// TIA Portal V17 export
// export: Created 2024-08-29T18:23:47.0171751Z, ExportSetting WithDefaults, DisplayName Totally Integrated Automation Portal, DisplayVersion V17 Update 7, DisplayName TIA Portal Openness, DisplayVersion V17 Update 7, DisplayName TIA Portal Version Control Interface, DisplayVersion V17, DisplayName SINAMICS Startdrive Advanced, DisplayVersion V17 SP2, DisplayName SINAMICS Startdrive G110M, G120, G120C, G120D, G120P, G115D, DisplayVersion V17 SP2, DisplayName SINAMICS Startdrive G130, G150, S120, S150, SINAMICS MV, S210, DisplayVersion V17 SP2, DisplayName STEP 7 Professional, DisplayVersion V17 Update 7, DisplayName STEP 7 Safety, DisplayVersion V17 Update 6, DisplayName WinCC Advanced / Unified PC, DisplayVersion V17 Update 7
FUNCTION "dintToBool" : Void   // FC10, LAD
{ S7_Optimized_Access := 'TRUE' }
VERSION : 0.1
// stored: AutoNumber true, IsIECCheckEnabled false, SetENOAutomatically false, UDAEnableTagReadback false
BEGIN

REGION Network 1: A INPUTS STATUS
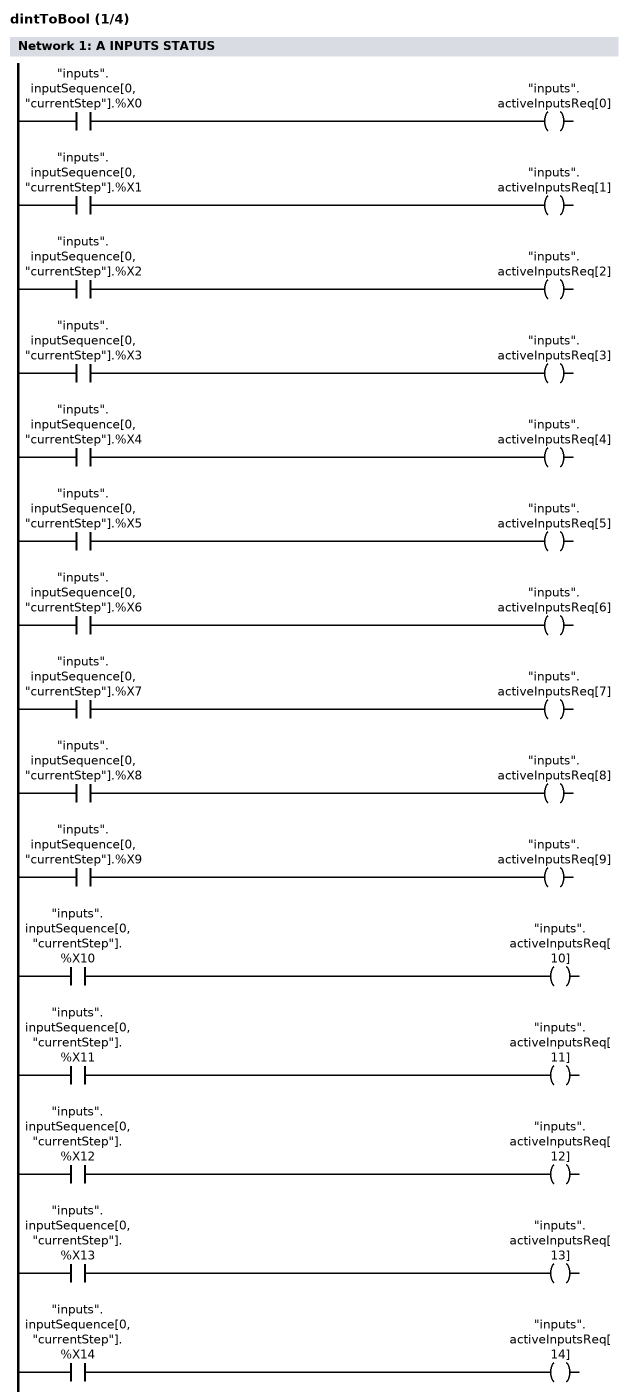
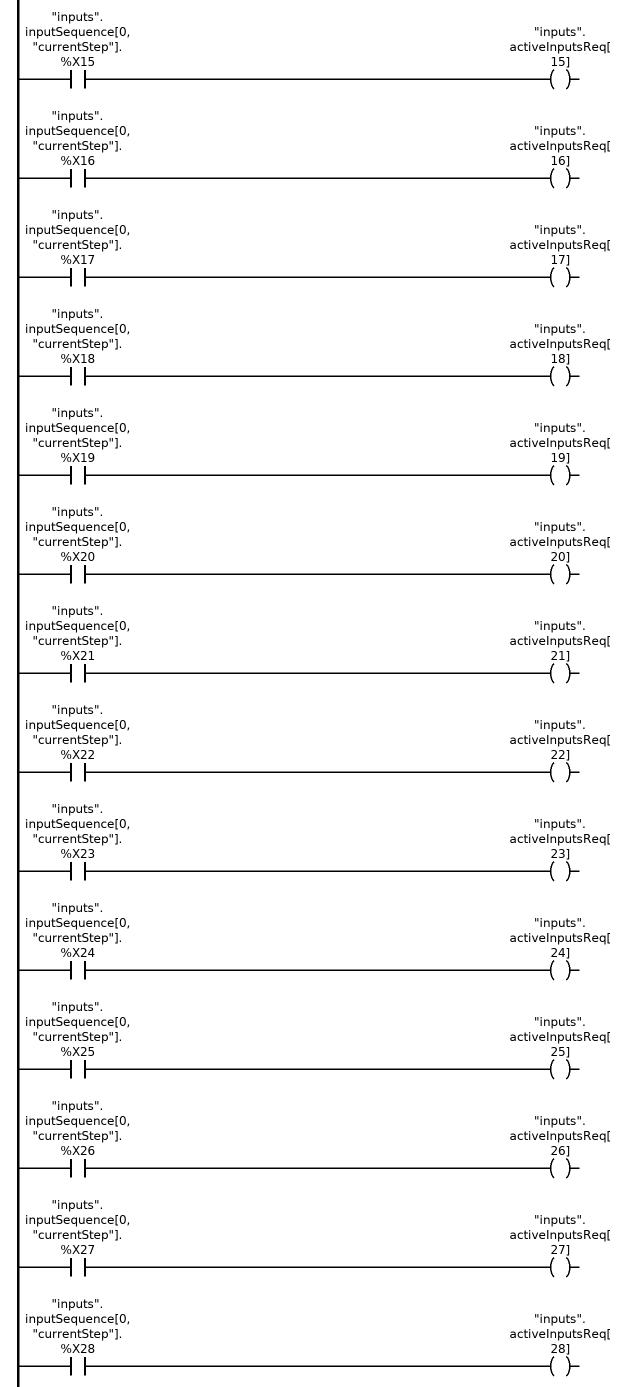
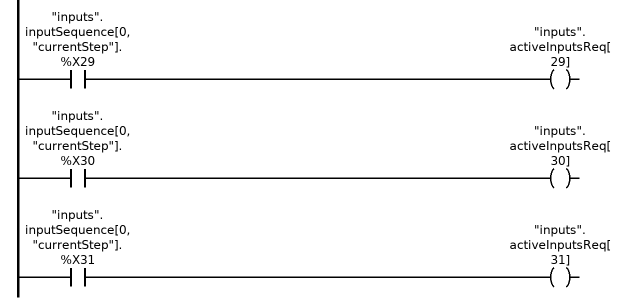
   RUNG wire#powerrail
      Contact( "inputs".inputSequence[0, "currentStep"].%X0 )
      Coil( "inputs".activeInputsReq[0] )
   END_RUNG
   RUNG wire#powerrail
      Contact( "inputs".inputSequence[0, "currentStep"].%X1 )
      Coil( "inputs".activeInputsReq[1] )
   END_RUNG
   RUNG wire#powerrail
      Contact( "inputs".inputSequence[0, "currentStep"].%X2 )
      Coil( "inputs".activeInputsReq[2] )
   END_RUNG
   RUNG wire#powerrail
      Contact( "inputs".inputSequence[0, "currentStep"].%X3 )
      Coil( "inputs".activeInputsReq[3] )
   END_RUNG
   RUNG wire#powerrail
      Contact( "inputs".inputSequence[0, "currentStep"].%X4 )
      Coil( "inputs".activeInputsReq[4] )
   END_RUNG
   RUNG wire#powerrail
      Contact( "inputs".inputSequence[0, "currentStep"].%X5 )
      Coil( "inputs".activeInputsReq[5] )
   END_RUNG
   RUNG wire#powerrail
      Contact( "inputs".inputSequence[0, "currentStep"].%X6 )
      Coil( "inputs".activeInputsReq[6] )
   END_RUNG
   RUNG wire#powerrail
      Contact( "inputs".inputSequence[0, "currentStep"].%X7 )
      Coil( "inputs".activeInputsReq[7] )
   END_RUNG
   RUNG wire#powerrail
      Contact( "inputs".inputSequence[0, "currentStep"].%X8 )
      Coil( "inputs".activeInputsReq[8] )
   END_RUNG
   RUNG wire#powerrail
      Contact( "inputs".inputSequence[0, "currentStep"].%X9 )
      Coil( "inputs".activeInputsReq[9] )
   END_RUNG
   RUNG wire#powerrail
      Contact( "inputs".inputSequence[0, "currentStep"].%X10 )
      Coil( "inputs".activeInputsReq[10] )
   END_RUNG
   RUNG wire#powerrail
      Contact( "inputs".inputSequence[0, "currentStep"].%X11 )
      Coil( "inputs".activeInputsReq[11] )
   END_RUNG
   RUNG wire#powerrail
      Contact( "inputs".inputSequence[0, "currentStep"].%X12 )
      Coil( "inputs".activeInputsReq[12] )
   END_RUNG
   RUNG wire#powerrail
      Contact( "inputs".inputSequence[0, "currentStep"].%X13 )
      Coil( "inputs".activeInputsReq[13] )
   END_RUNG
   RUNG wire#powerrail
      Contact( "inputs".inputSequence[0, "currentStep"].%X14 )
      Coil( "inputs".activeInputsReq[14] )
   END_RUNG
   RUNG wire#powerrail
      Contact( "inputs".inputSequence[0, "currentStep"].%X15 )
      Coil( "inputs".activeInputsReq[15] )
   END_RUNG
   RUNG wire#powerrail
      Contact( "inputs".inputSequence[0, "currentStep"].%X16 )
      Coil( "inputs".activeInputsReq[16] )
   END_RUNG
   RUNG wire#powerrail
      Contact( "inputs".inputSequence[0, "currentStep"].%X17 )
      Coil( "inputs".activeInputsReq[17] )
   END_RUNG
   RUNG wire#powerrail
      Contact( "inputs".inputSequence[0, "currentStep"].%X18 )
      Coil( "inputs".activeInputsReq[18] )
   END_RUNG
   RUNG wire#powerrail
      Contact( "inputs".inputSequence[0, "currentStep"].%X19 )
      Coil( "inputs".activeInputsReq[19] )
   END_RUNG
   RUNG wire#powerrail
      Contact( "inputs".inputSequence[0, "currentStep"].%X20 )
      Coil( "inputs".activeInputsReq[20] )
   END_RUNG
   RUNG wire#powerrail
      Contact( "inputs".inputSequence[0, "currentStep"].%X21 )
      Coil( "inputs".activeInputsReq[21] )
   END_RUNG
   RUNG wire#powerrail
      Contact( "inputs".inputSequence[0, "currentStep"].%X22 )
      Coil( "inputs".activeInputsReq[22] )
   END_RUNG
   RUNG wire#powerrail
      Contact( "inputs".inputSequence[0, "currentStep"].%X23 )
      Coil( "inputs".activeInputsReq[23] )
   END_RUNG
   RUNG wire#powerrail
      Contact( "inputs".inputSequence[0, "currentStep"].%X24 )
      Coil( "inputs".activeInputsReq[24] )
   END_RUNG
   RUNG wire#powerrail
      Contact( "inputs".inputSequence[0, "currentStep"].%X25 )
      Coil( "inputs".activeInputsReq[25] )
   END_RUNG
   RUNG wire#powerrail
      Contact( "inputs".inputSequence[0, "currentStep"].%X26 )
      Coil( "inputs".activeInputsReq[26] )
   END_RUNG
   RUNG wire#powerrail
      Contact( "inputs".inputSequence[0, "currentStep"].%X27 )
      Coil( "inputs".activeInputsReq[27] )
   END_RUNG
   RUNG wire#powerrail
      Contact( "inputs".inputSequence[0, "currentStep"].%X28 )
      Coil( "inputs".activeInputsReq[28] )
   END_RUNG
   RUNG wire#powerrail
      Contact( "inputs".inputSequence[0, "currentStep"].%X29 )
      Coil( "inputs".activeInputsReq[29] )
   END_RUNG
   RUNG wire#powerrail
      Contact( "inputs".inputSequence[0, "currentStep"].%X30 )
      Coil( "inputs".activeInputsReq[30] )
   END_RUNG
   RUNG wire#powerrail
      Contact( "inputs".inputSequence[0, "currentStep"].%X31 )
      Coil( "inputs".activeInputsReq[31] )
   END_RUNG
   // the same network as SCL:
   "inputs".activeInputsReq[0] := "inputs".inputSequence[0, "currentStep"].%X0;
   "inputs".activeInputsReq[1] := "inputs".inputSequence[0, "currentStep"].%X1;
   "inputs".activeInputsReq[2] := "inputs".inputSequence[0, "currentStep"].%X2;
   "inputs".activeInputsReq[3] := "inputs".inputSequence[0, "currentStep"].%X3;
   "inputs".activeInputsReq[4] := "inputs".inputSequence[0, "currentStep"].%X4;
   "inputs".activeInputsReq[5] := "inputs".inputSequence[0, "currentStep"].%X5;
   "inputs".activeInputsReq[6] := "inputs".inputSequence[0, "currentStep"].%X6;
   "inputs".activeInputsReq[7] := "inputs".inputSequence[0, "currentStep"].%X7;
   "inputs".activeInputsReq[8] := "inputs".inputSequence[0, "currentStep"].%X8;
   "inputs".activeInputsReq[9] := "inputs".inputSequence[0, "currentStep"].%X9;
   "inputs".activeInputsReq[10] := "inputs".inputSequence[0, "currentStep"].%X10;
   "inputs".activeInputsReq[11] := "inputs".inputSequence[0, "currentStep"].%X11;
   "inputs".activeInputsReq[12] := "inputs".inputSequence[0, "currentStep"].%X12;
   "inputs".activeInputsReq[13] := "inputs".inputSequence[0, "currentStep"].%X13;
   "inputs".activeInputsReq[14] := "inputs".inputSequence[0, "currentStep"].%X14;
   "inputs".activeInputsReq[15] := "inputs".inputSequence[0, "currentStep"].%X15;
   "inputs".activeInputsReq[16] := "inputs".inputSequence[0, "currentStep"].%X16;
   "inputs".activeInputsReq[17] := "inputs".inputSequence[0, "currentStep"].%X17;
   "inputs".activeInputsReq[18] := "inputs".inputSequence[0, "currentStep"].%X18;
   "inputs".activeInputsReq[19] := "inputs".inputSequence[0, "currentStep"].%X19;
   "inputs".activeInputsReq[20] := "inputs".inputSequence[0, "currentStep"].%X20;
   "inputs".activeInputsReq[21] := "inputs".inputSequence[0, "currentStep"].%X21;
   "inputs".activeInputsReq[22] := "inputs".inputSequence[0, "currentStep"].%X22;
   "inputs".activeInputsReq[23] := "inputs".inputSequence[0, "currentStep"].%X23;
   "inputs".activeInputsReq[24] := "inputs".inputSequence[0, "currentStep"].%X24;
   "inputs".activeInputsReq[25] := "inputs".inputSequence[0, "currentStep"].%X25;
   "inputs".activeInputsReq[26] := "inputs".inputSequence[0, "currentStep"].%X26;
   "inputs".activeInputsReq[27] := "inputs".inputSequence[0, "currentStep"].%X27;
   "inputs".activeInputsReq[28] := "inputs".inputSequence[0, "currentStep"].%X28;
   "inputs".activeInputsReq[29] := "inputs".inputSequence[0, "currentStep"].%X29;
   "inputs".activeInputsReq[30] := "inputs".inputSequence[0, "currentStep"].%X30;
   "inputs".activeInputsReq[31] := "inputs".inputSequence[0, "currentStep"].%X31;
END_REGION

REGION Network 2: MASK INPUTS STATUS
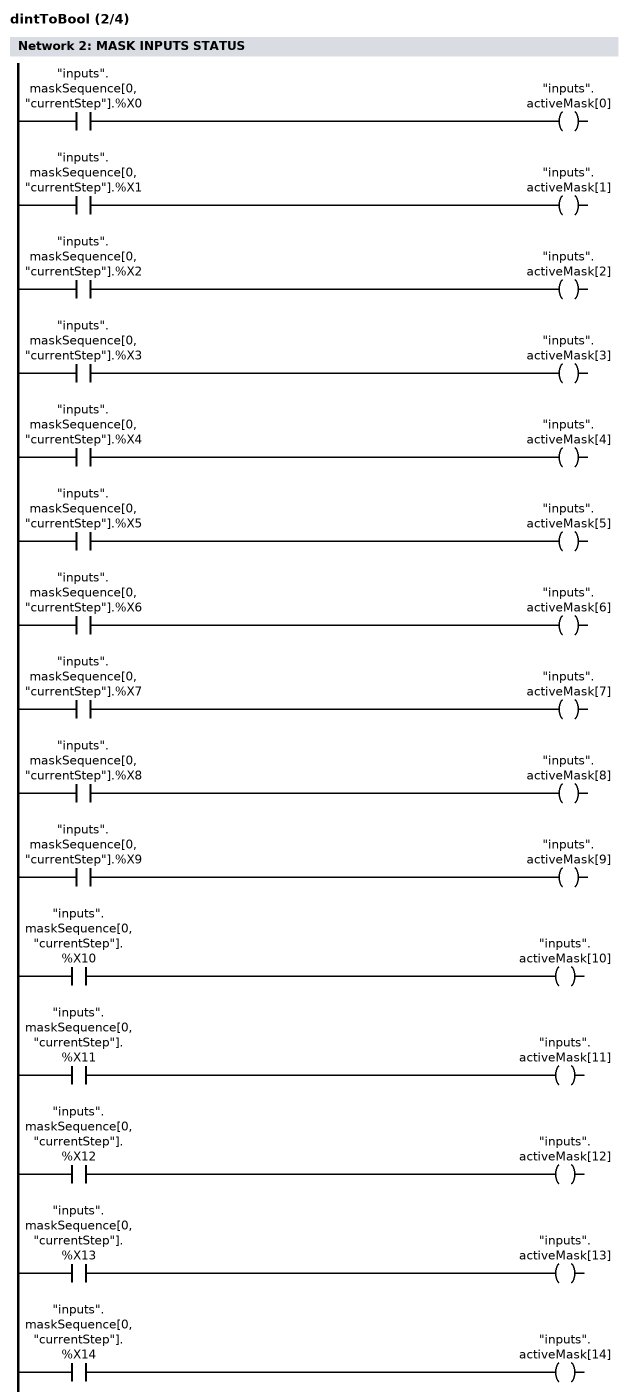
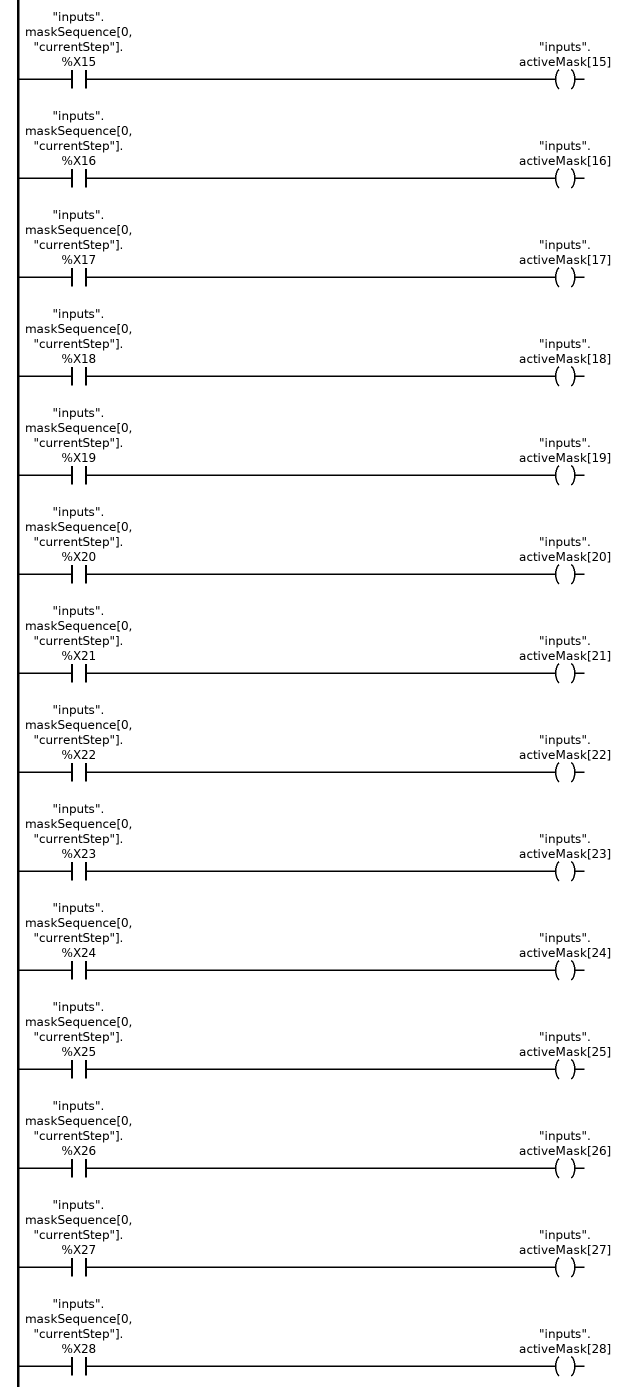
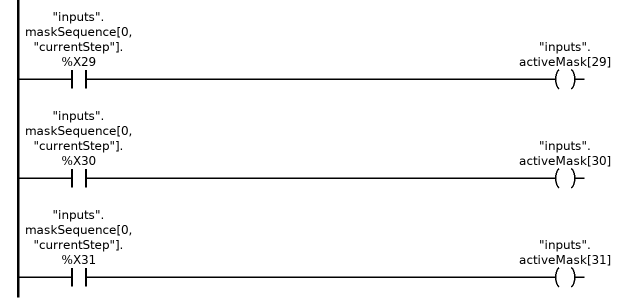
   RUNG wire#powerrail
      Contact( "inputs".maskSequence[0, "currentStep"].%X0 )
      Coil( "inputs".activeMask[0] )
   END_RUNG
   RUNG wire#powerrail
      Contact( "inputs".maskSequence[0, "currentStep"].%X1 )
      Coil( "inputs".activeMask[1] )
   END_RUNG
   RUNG wire#powerrail
      Contact( "inputs".maskSequence[0, "currentStep"].%X2 )
      Coil( "inputs".activeMask[2] )
   END_RUNG
   RUNG wire#powerrail
      Contact( "inputs".maskSequence[0, "currentStep"].%X3 )
      Coil( "inputs".activeMask[3] )
   END_RUNG
   RUNG wire#powerrail
      Contact( "inputs".maskSequence[0, "currentStep"].%X4 )
      Coil( "inputs".activeMask[4] )
   END_RUNG
   RUNG wire#powerrail
      Contact( "inputs".maskSequence[0, "currentStep"].%X5 )
      Coil( "inputs".activeMask[5] )
   END_RUNG
   RUNG wire#powerrail
      Contact( "inputs".maskSequence[0, "currentStep"].%X6 )
      Coil( "inputs".activeMask[6] )
   END_RUNG
   RUNG wire#powerrail
      Contact( "inputs".maskSequence[0, "currentStep"].%X7 )
      Coil( "inputs".activeMask[7] )
   END_RUNG
   RUNG wire#powerrail
      Contact( "inputs".maskSequence[0, "currentStep"].%X8 )
      Coil( "inputs".activeMask[8] )
   END_RUNG
   RUNG wire#powerrail
      Contact( "inputs".maskSequence[0, "currentStep"].%X9 )
      Coil( "inputs".activeMask[9] )
   END_RUNG
   RUNG wire#powerrail
      Contact( "inputs".maskSequence[0, "currentStep"].%X10 )
      Coil( "inputs".activeMask[10] )
   END_RUNG
   RUNG wire#powerrail
      Contact( "inputs".maskSequence[0, "currentStep"].%X11 )
      Coil( "inputs".activeMask[11] )
   END_RUNG
   RUNG wire#powerrail
      Contact( "inputs".maskSequence[0, "currentStep"].%X12 )
      Coil( "inputs".activeMask[12] )
   END_RUNG
   RUNG wire#powerrail
      Contact( "inputs".maskSequence[0, "currentStep"].%X13 )
      Coil( "inputs".activeMask[13] )
   END_RUNG
   RUNG wire#powerrail
      Contact( "inputs".maskSequence[0, "currentStep"].%X14 )
      Coil( "inputs".activeMask[14] )
   END_RUNG
   RUNG wire#powerrail
      Contact( "inputs".maskSequence[0, "currentStep"].%X15 )
      Coil( "inputs".activeMask[15] )
   END_RUNG
   RUNG wire#powerrail
      Contact( "inputs".maskSequence[0, "currentStep"].%X16 )
      Coil( "inputs".activeMask[16] )
   END_RUNG
   RUNG wire#powerrail
      Contact( "inputs".maskSequence[0, "currentStep"].%X17 )
      Coil( "inputs".activeMask[17] )
   END_RUNG
   RUNG wire#powerrail
      Contact( "inputs".maskSequence[0, "currentStep"].%X18 )
      Coil( "inputs".activeMask[18] )
   END_RUNG
   RUNG wire#powerrail
      Contact( "inputs".maskSequence[0, "currentStep"].%X19 )
      Coil( "inputs".activeMask[19] )
   END_RUNG
   RUNG wire#powerrail
      Contact( "inputs".maskSequence[0, "currentStep"].%X20 )
      Coil( "inputs".activeMask[20] )
   END_RUNG
   RUNG wire#powerrail
      Contact( "inputs".maskSequence[0, "currentStep"].%X21 )
      Coil( "inputs".activeMask[21] )
   END_RUNG
   RUNG wire#powerrail
      Contact( "inputs".maskSequence[0, "currentStep"].%X22 )
      Coil( "inputs".activeMask[22] )
   END_RUNG
   RUNG wire#powerrail
      Contact( "inputs".maskSequence[0, "currentStep"].%X23 )
      Coil( "inputs".activeMask[23] )
   END_RUNG
   RUNG wire#powerrail
      Contact( "inputs".maskSequence[0, "currentStep"].%X24 )
      Coil( "inputs".activeMask[24] )
   END_RUNG
   RUNG wire#powerrail
      Contact( "inputs".maskSequence[0, "currentStep"].%X25 )
      Coil( "inputs".activeMask[25] )
   END_RUNG
   RUNG wire#powerrail
      Contact( "inputs".maskSequence[0, "currentStep"].%X26 )
      Coil( "inputs".activeMask[26] )
   END_RUNG
   RUNG wire#powerrail
      Contact( "inputs".maskSequence[0, "currentStep"].%X27 )
      Coil( "inputs".activeMask[27] )
   END_RUNG
   RUNG wire#powerrail
      Contact( "inputs".maskSequence[0, "currentStep"].%X28 )
      Coil( "inputs".activeMask[28] )
   END_RUNG
   RUNG wire#powerrail
      Contact( "inputs".maskSequence[0, "currentStep"].%X29 )
      Coil( "inputs".activeMask[29] )
   END_RUNG
   RUNG wire#powerrail
      Contact( "inputs".maskSequence[0, "currentStep"].%X30 )
      Coil( "inputs".activeMask[30] )
   END_RUNG
   RUNG wire#powerrail
      Contact( "inputs".maskSequence[0, "currentStep"].%X31 )
      Coil( "inputs".activeMask[31] )
   END_RUNG
   // the same network as SCL:
   "inputs".activeMask[0] := "inputs".maskSequence[0, "currentStep"].%X0;
   "inputs".activeMask[1] := "inputs".maskSequence[0, "currentStep"].%X1;
   "inputs".activeMask[2] := "inputs".maskSequence[0, "currentStep"].%X2;
   "inputs".activeMask[3] := "inputs".maskSequence[0, "currentStep"].%X3;
   "inputs".activeMask[4] := "inputs".maskSequence[0, "currentStep"].%X4;
   "inputs".activeMask[5] := "inputs".maskSequence[0, "currentStep"].%X5;
   "inputs".activeMask[6] := "inputs".maskSequence[0, "currentStep"].%X6;
   "inputs".activeMask[7] := "inputs".maskSequence[0, "currentStep"].%X7;
   "inputs".activeMask[8] := "inputs".maskSequence[0, "currentStep"].%X8;
   "inputs".activeMask[9] := "inputs".maskSequence[0, "currentStep"].%X9;
   "inputs".activeMask[10] := "inputs".maskSequence[0, "currentStep"].%X10;
   "inputs".activeMask[11] := "inputs".maskSequence[0, "currentStep"].%X11;
   "inputs".activeMask[12] := "inputs".maskSequence[0, "currentStep"].%X12;
   "inputs".activeMask[13] := "inputs".maskSequence[0, "currentStep"].%X13;
   "inputs".activeMask[14] := "inputs".maskSequence[0, "currentStep"].%X14;
   "inputs".activeMask[15] := "inputs".maskSequence[0, "currentStep"].%X15;
   "inputs".activeMask[16] := "inputs".maskSequence[0, "currentStep"].%X16;
   "inputs".activeMask[17] := "inputs".maskSequence[0, "currentStep"].%X17;
   "inputs".activeMask[18] := "inputs".maskSequence[0, "currentStep"].%X18;
   "inputs".activeMask[19] := "inputs".maskSequence[0, "currentStep"].%X19;
   "inputs".activeMask[20] := "inputs".maskSequence[0, "currentStep"].%X20;
   "inputs".activeMask[21] := "inputs".maskSequence[0, "currentStep"].%X21;
   "inputs".activeMask[22] := "inputs".maskSequence[0, "currentStep"].%X22;
   "inputs".activeMask[23] := "inputs".maskSequence[0, "currentStep"].%X23;
   "inputs".activeMask[24] := "inputs".maskSequence[0, "currentStep"].%X24;
   "inputs".activeMask[25] := "inputs".maskSequence[0, "currentStep"].%X25;
   "inputs".activeMask[26] := "inputs".maskSequence[0, "currentStep"].%X26;
   "inputs".activeMask[27] := "inputs".maskSequence[0, "currentStep"].%X27;
   "inputs".activeMask[28] := "inputs".maskSequence[0, "currentStep"].%X28;
   "inputs".activeMask[29] := "inputs".maskSequence[0, "currentStep"].%X29;
   "inputs".activeMask[30] := "inputs".maskSequence[0, "currentStep"].%X30;
   "inputs".activeMask[31] := "inputs".maskSequence[0, "currentStep"].%X31;
END_REGION

REGION Network 3: B OUTPUTS STATUS
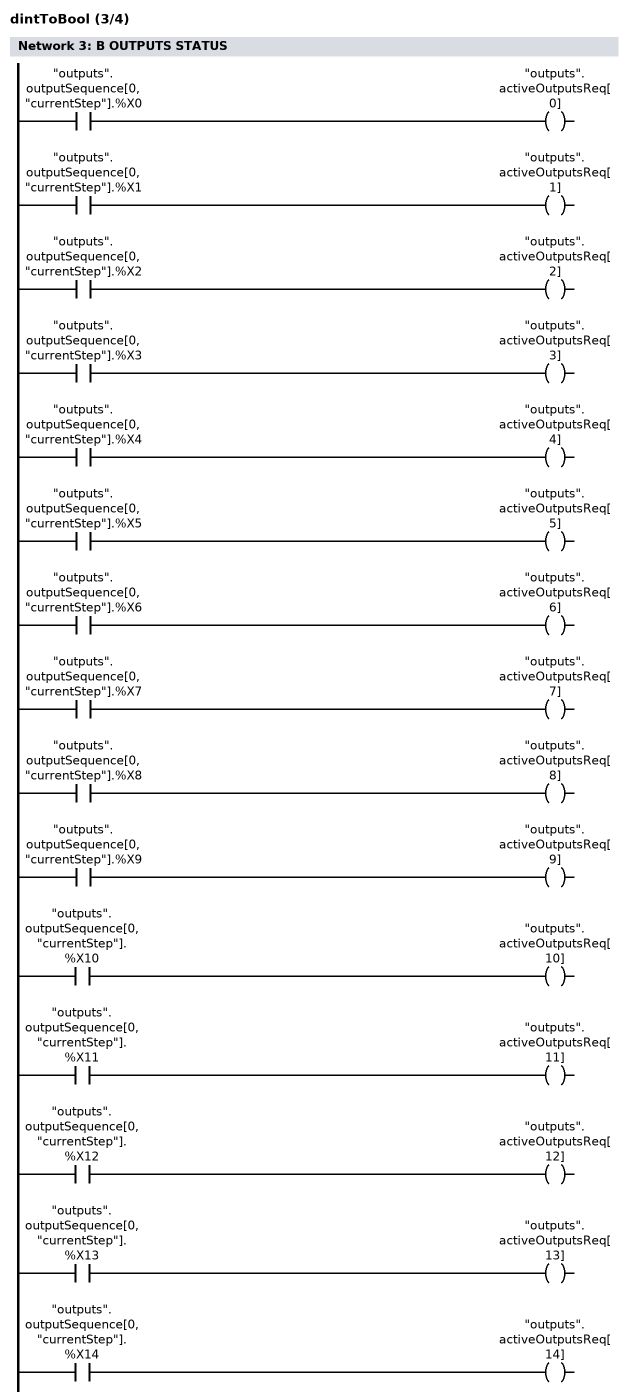
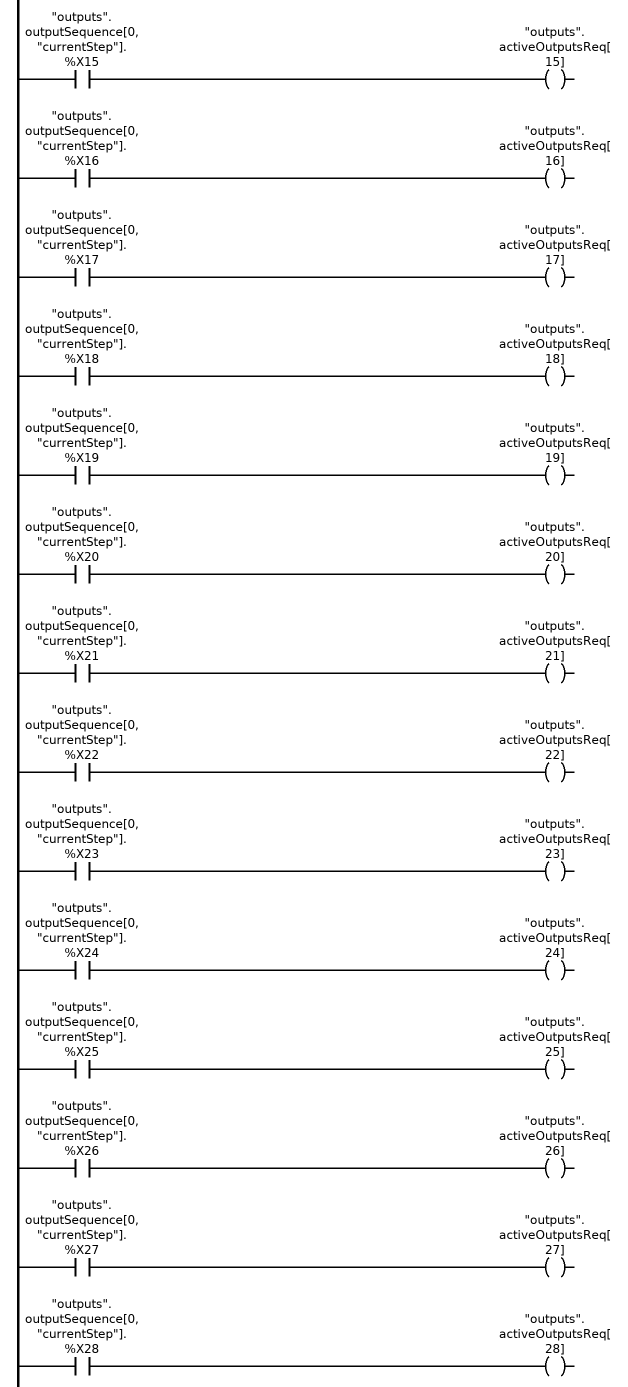
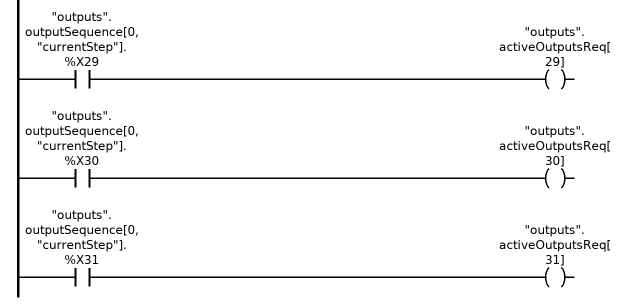
   RUNG wire#powerrail
      Contact( "outputs".outputSequence[0, "currentStep"].%X0 )
      Coil( "outputs".activeOutputsReq[0] )
   END_RUNG
   RUNG wire#powerrail
      Contact( "outputs".outputSequence[0, "currentStep"].%X1 )
      Coil( "outputs".activeOutputsReq[1] )
   END_RUNG
   RUNG wire#powerrail
      Contact( "outputs".outputSequence[0, "currentStep"].%X2 )
      Coil( "outputs".activeOutputsReq[2] )
   END_RUNG
   RUNG wire#powerrail
      Contact( "outputs".outputSequence[0, "currentStep"].%X3 )
      Coil( "outputs".activeOutputsReq[3] )
   END_RUNG
   RUNG wire#powerrail
      Contact( "outputs".outputSequence[0, "currentStep"].%X4 )
      Coil( "outputs".activeOutputsReq[4] )
   END_RUNG
   RUNG wire#powerrail
      Contact( "outputs".outputSequence[0, "currentStep"].%X5 )
      Coil( "outputs".activeOutputsReq[5] )
   END_RUNG
   RUNG wire#powerrail
      Contact( "outputs".outputSequence[0, "currentStep"].%X6 )
      Coil( "outputs".activeOutputsReq[6] )
   END_RUNG
   RUNG wire#powerrail
      Contact( "outputs".outputSequence[0, "currentStep"].%X7 )
      Coil( "outputs".activeOutputsReq[7] )
   END_RUNG
   RUNG wire#powerrail
      Contact( "outputs".outputSequence[0, "currentStep"].%X8 )
      Coil( "outputs".activeOutputsReq[8] )
   END_RUNG
   RUNG wire#powerrail
      Contact( "outputs".outputSequence[0, "currentStep"].%X9 )
      Coil( "outputs".activeOutputsReq[9] )
   END_RUNG
   RUNG wire#powerrail
      Contact( "outputs".outputSequence[0, "currentStep"].%X10 )
      Coil( "outputs".activeOutputsReq[10] )
   END_RUNG
   RUNG wire#powerrail
      Contact( "outputs".outputSequence[0, "currentStep"].%X11 )
      Coil( "outputs".activeOutputsReq[11] )
   END_RUNG
   RUNG wire#powerrail
      Contact( "outputs".outputSequence[0, "currentStep"].%X12 )
      Coil( "outputs".activeOutputsReq[12] )
   END_RUNG
   RUNG wire#powerrail
      Contact( "outputs".outputSequence[0, "currentStep"].%X13 )
      Coil( "outputs".activeOutputsReq[13] )
   END_RUNG
   RUNG wire#powerrail
      Contact( "outputs".outputSequence[0, "currentStep"].%X14 )
      Coil( "outputs".activeOutputsReq[14] )
   END_RUNG
   RUNG wire#powerrail
      Contact( "outputs".outputSequence[0, "currentStep"].%X15 )
      Coil( "outputs".activeOutputsReq[15] )
   END_RUNG
   RUNG wire#powerrail
      Contact( "outputs".outputSequence[0, "currentStep"].%X16 )
      Coil( "outputs".activeOutputsReq[16] )
   END_RUNG
   RUNG wire#powerrail
      Contact( "outputs".outputSequence[0, "currentStep"].%X17 )
      Coil( "outputs".activeOutputsReq[17] )
   END_RUNG
   RUNG wire#powerrail
      Contact( "outputs".outputSequence[0, "currentStep"].%X18 )
      Coil( "outputs".activeOutputsReq[18] )
   END_RUNG
   RUNG wire#powerrail
      Contact( "outputs".outputSequence[0, "currentStep"].%X19 )
      Coil( "outputs".activeOutputsReq[19] )
   END_RUNG
   RUNG wire#powerrail
      Contact( "outputs".outputSequence[0, "currentStep"].%X20 )
      Coil( "outputs".activeOutputsReq[20] )
   END_RUNG
   RUNG wire#powerrail
      Contact( "outputs".outputSequence[0, "currentStep"].%X21 )
      Coil( "outputs".activeOutputsReq[21] )
   END_RUNG
   RUNG wire#powerrail
      Contact( "outputs".outputSequence[0, "currentStep"].%X22 )
      Coil( "outputs".activeOutputsReq[22] )
   END_RUNG
   RUNG wire#powerrail
      Contact( "outputs".outputSequence[0, "currentStep"].%X23 )
      Coil( "outputs".activeOutputsReq[23] )
   END_RUNG
   RUNG wire#powerrail
      Contact( "outputs".outputSequence[0, "currentStep"].%X24 )
      Coil( "outputs".activeOutputsReq[24] )
   END_RUNG
   RUNG wire#powerrail
      Contact( "outputs".outputSequence[0, "currentStep"].%X25 )
      Coil( "outputs".activeOutputsReq[25] )
   END_RUNG
   RUNG wire#powerrail
      Contact( "outputs".outputSequence[0, "currentStep"].%X26 )
      Coil( "outputs".activeOutputsReq[26] )
   END_RUNG
   RUNG wire#powerrail
      Contact( "outputs".outputSequence[0, "currentStep"].%X27 )
      Coil( "outputs".activeOutputsReq[27] )
   END_RUNG
   RUNG wire#powerrail
      Contact( "outputs".outputSequence[0, "currentStep"].%X28 )
      Coil( "outputs".activeOutputsReq[28] )
   END_RUNG
   RUNG wire#powerrail
      Contact( "outputs".outputSequence[0, "currentStep"].%X29 )
      Coil( "outputs".activeOutputsReq[29] )
   END_RUNG
   RUNG wire#powerrail
      Contact( "outputs".outputSequence[0, "currentStep"].%X30 )
      Coil( "outputs".activeOutputsReq[30] )
   END_RUNG
   RUNG wire#powerrail
      Contact( "outputs".outputSequence[0, "currentStep"].%X31 )
      Coil( "outputs".activeOutputsReq[31] )
   END_RUNG
   // the same network as SCL:
   "outputs".activeOutputsReq[0] := "outputs".outputSequence[0, "currentStep"].%X0;
   "outputs".activeOutputsReq[1] := "outputs".outputSequence[0, "currentStep"].%X1;
   "outputs".activeOutputsReq[2] := "outputs".outputSequence[0, "currentStep"].%X2;
   "outputs".activeOutputsReq[3] := "outputs".outputSequence[0, "currentStep"].%X3;
   "outputs".activeOutputsReq[4] := "outputs".outputSequence[0, "currentStep"].%X4;
   "outputs".activeOutputsReq[5] := "outputs".outputSequence[0, "currentStep"].%X5;
   "outputs".activeOutputsReq[6] := "outputs".outputSequence[0, "currentStep"].%X6;
   "outputs".activeOutputsReq[7] := "outputs".outputSequence[0, "currentStep"].%X7;
   "outputs".activeOutputsReq[8] := "outputs".outputSequence[0, "currentStep"].%X8;
   "outputs".activeOutputsReq[9] := "outputs".outputSequence[0, "currentStep"].%X9;
   "outputs".activeOutputsReq[10] := "outputs".outputSequence[0, "currentStep"].%X10;
   "outputs".activeOutputsReq[11] := "outputs".outputSequence[0, "currentStep"].%X11;
   "outputs".activeOutputsReq[12] := "outputs".outputSequence[0, "currentStep"].%X12;
   "outputs".activeOutputsReq[13] := "outputs".outputSequence[0, "currentStep"].%X13;
   "outputs".activeOutputsReq[14] := "outputs".outputSequence[0, "currentStep"].%X14;
   "outputs".activeOutputsReq[15] := "outputs".outputSequence[0, "currentStep"].%X15;
   "outputs".activeOutputsReq[16] := "outputs".outputSequence[0, "currentStep"].%X16;
   "outputs".activeOutputsReq[17] := "outputs".outputSequence[0, "currentStep"].%X17;
   "outputs".activeOutputsReq[18] := "outputs".outputSequence[0, "currentStep"].%X18;
   "outputs".activeOutputsReq[19] := "outputs".outputSequence[0, "currentStep"].%X19;
   "outputs".activeOutputsReq[20] := "outputs".outputSequence[0, "currentStep"].%X20;
   "outputs".activeOutputsReq[21] := "outputs".outputSequence[0, "currentStep"].%X21;
   "outputs".activeOutputsReq[22] := "outputs".outputSequence[0, "currentStep"].%X22;
   "outputs".activeOutputsReq[23] := "outputs".outputSequence[0, "currentStep"].%X23;
   "outputs".activeOutputsReq[24] := "outputs".outputSequence[0, "currentStep"].%X24;
   "outputs".activeOutputsReq[25] := "outputs".outputSequence[0, "currentStep"].%X25;
   "outputs".activeOutputsReq[26] := "outputs".outputSequence[0, "currentStep"].%X26;
   "outputs".activeOutputsReq[27] := "outputs".outputSequence[0, "currentStep"].%X27;
   "outputs".activeOutputsReq[28] := "outputs".outputSequence[0, "currentStep"].%X28;
   "outputs".activeOutputsReq[29] := "outputs".outputSequence[0, "currentStep"].%X29;
   "outputs".activeOutputsReq[30] := "outputs".outputSequence[0, "currentStep"].%X30;
   "outputs".activeOutputsReq[31] := "outputs".outputSequence[0, "currentStep"].%X31;
END_REGION

REGION Network 4: MASK OUTPUTS STATUS
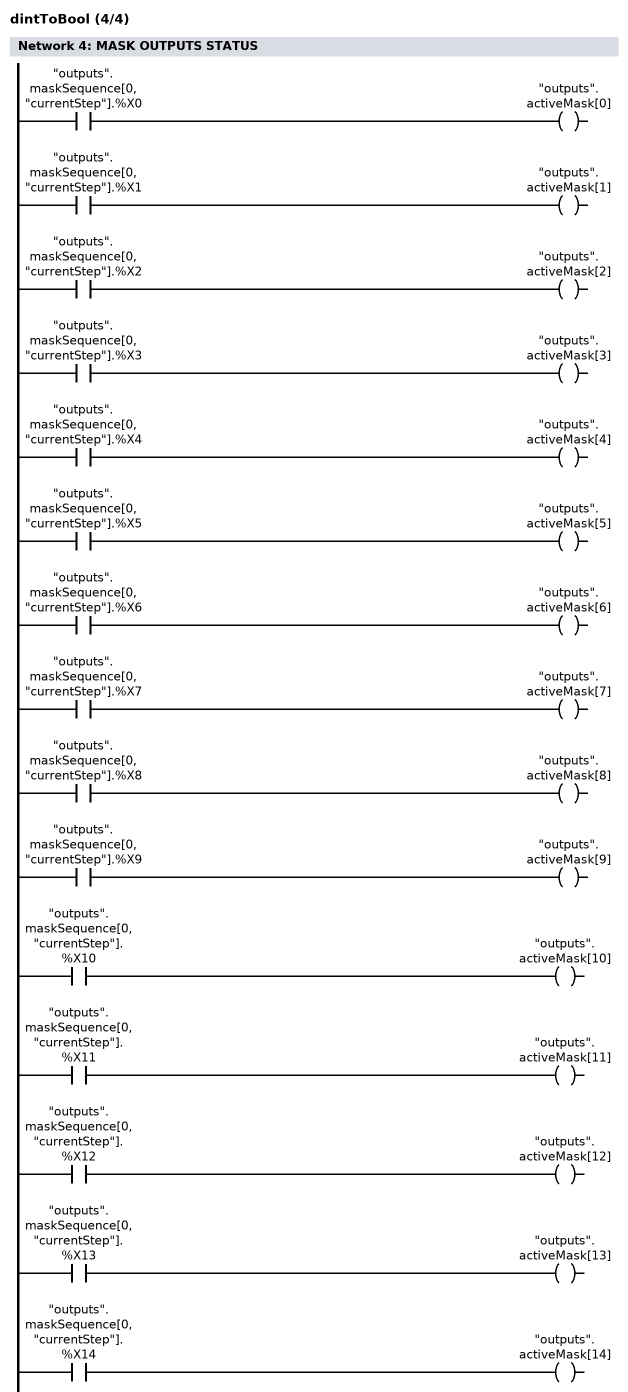
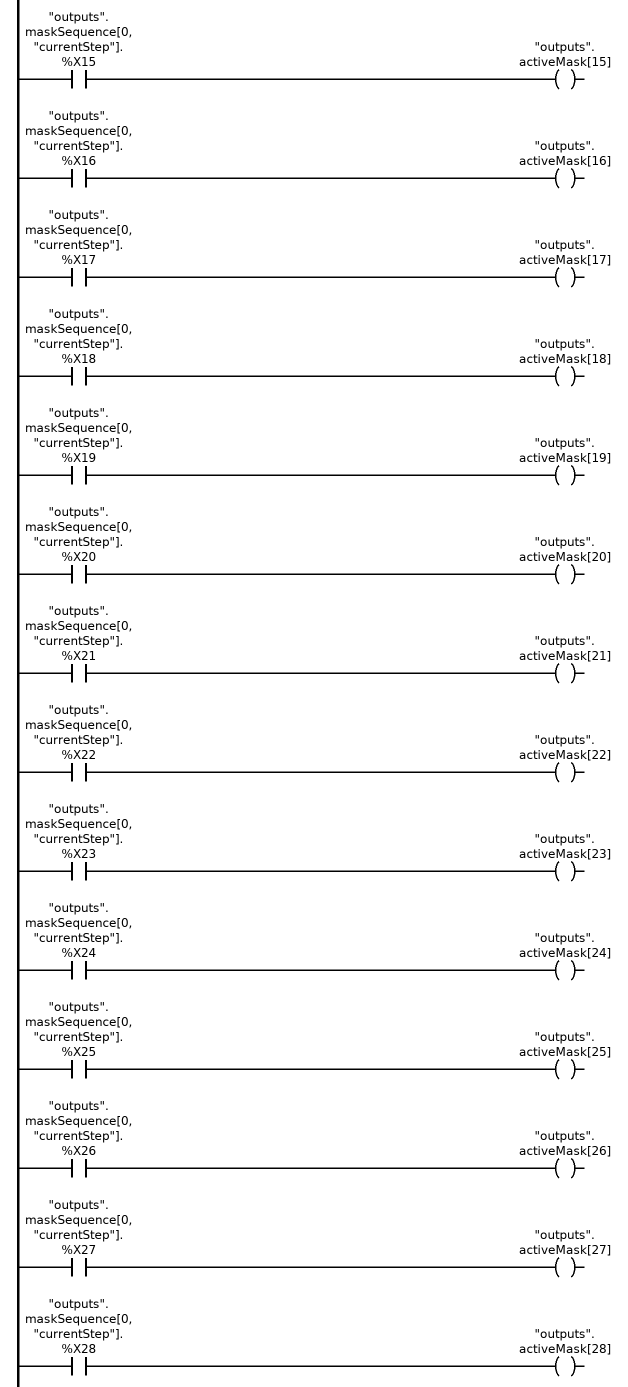
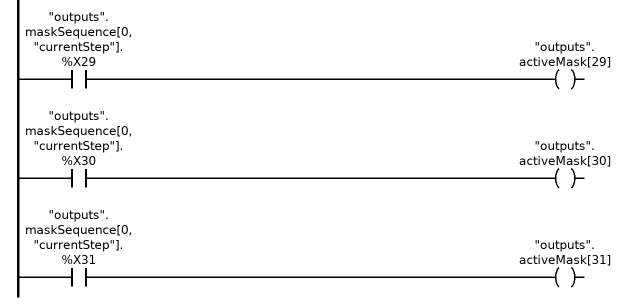
   RUNG wire#powerrail
      Contact( "outputs".maskSequence[0, "currentStep"].%X0 )
      Coil( "outputs".activeMask[0] )
   END_RUNG
   RUNG wire#powerrail
      Contact( "outputs".maskSequence[0, "currentStep"].%X1 )
      Coil( "outputs".activeMask[1] )
   END_RUNG
   RUNG wire#powerrail
      Contact( "outputs".maskSequence[0, "currentStep"].%X2 )
      Coil( "outputs".activeMask[2] )
   END_RUNG
   RUNG wire#powerrail
      Contact( "outputs".maskSequence[0, "currentStep"].%X3 )
      Coil( "outputs".activeMask[3] )
   END_RUNG
   RUNG wire#powerrail
      Contact( "outputs".maskSequence[0, "currentStep"].%X4 )
      Coil( "outputs".activeMask[4] )
   END_RUNG
   RUNG wire#powerrail
      Contact( "outputs".maskSequence[0, "currentStep"].%X5 )
      Coil( "outputs".activeMask[5] )
   END_RUNG
   RUNG wire#powerrail
      Contact( "outputs".maskSequence[0, "currentStep"].%X6 )
      Coil( "outputs".activeMask[6] )
   END_RUNG
   RUNG wire#powerrail
      Contact( "outputs".maskSequence[0, "currentStep"].%X7 )
      Coil( "outputs".activeMask[7] )
   END_RUNG
   RUNG wire#powerrail
      Contact( "outputs".maskSequence[0, "currentStep"].%X8 )
      Coil( "outputs".activeMask[8] )
   END_RUNG
   RUNG wire#powerrail
      Contact( "outputs".maskSequence[0, "currentStep"].%X9 )
      Coil( "outputs".activeMask[9] )
   END_RUNG
   RUNG wire#powerrail
      Contact( "outputs".maskSequence[0, "currentStep"].%X10 )
      Coil( "outputs".activeMask[10] )
   END_RUNG
   RUNG wire#powerrail
      Contact( "outputs".maskSequence[0, "currentStep"].%X11 )
      Coil( "outputs".activeMask[11] )
   END_RUNG
   RUNG wire#powerrail
      Contact( "outputs".maskSequence[0, "currentStep"].%X12 )
      Coil( "outputs".activeMask[12] )
   END_RUNG
   RUNG wire#powerrail
      Contact( "outputs".maskSequence[0, "currentStep"].%X13 )
      Coil( "outputs".activeMask[13] )
   END_RUNG
   RUNG wire#powerrail
      Contact( "outputs".maskSequence[0, "currentStep"].%X14 )
      Coil( "outputs".activeMask[14] )
   END_RUNG
   RUNG wire#powerrail
      Contact( "outputs".maskSequence[0, "currentStep"].%X15 )
      Coil( "outputs".activeMask[15] )
   END_RUNG
   RUNG wire#powerrail
      Contact( "outputs".maskSequence[0, "currentStep"].%X16 )
      Coil( "outputs".activeMask[16] )
   END_RUNG
   RUNG wire#powerrail
      Contact( "outputs".maskSequence[0, "currentStep"].%X17 )
      Coil( "outputs".activeMask[17] )
   END_RUNG
   RUNG wire#powerrail
      Contact( "outputs".maskSequence[0, "currentStep"].%X18 )
      Coil( "outputs".activeMask[18] )
   END_RUNG
   RUNG wire#powerrail
      Contact( "outputs".maskSequence[0, "currentStep"].%X19 )
      Coil( "outputs".activeMask[19] )
   END_RUNG
   RUNG wire#powerrail
      Contact( "outputs".maskSequence[0, "currentStep"].%X20 )
      Coil( "outputs".activeMask[20] )
   END_RUNG
   RUNG wire#powerrail
      Contact( "outputs".maskSequence[0, "currentStep"].%X21 )
      Coil( "outputs".activeMask[21] )
   END_RUNG
   RUNG wire#powerrail
      Contact( "outputs".maskSequence[0, "currentStep"].%X22 )
      Coil( "outputs".activeMask[22] )
   END_RUNG
   RUNG wire#powerrail
      Contact( "outputs".maskSequence[0, "currentStep"].%X23 )
      Coil( "outputs".activeMask[23] )
   END_RUNG
   RUNG wire#powerrail
      Contact( "outputs".maskSequence[0, "currentStep"].%X24 )
      Coil( "outputs".activeMask[24] )
   END_RUNG
   RUNG wire#powerrail
      Contact( "outputs".maskSequence[0, "currentStep"].%X25 )
      Coil( "outputs".activeMask[25] )
   END_RUNG
   RUNG wire#powerrail
      Contact( "outputs".maskSequence[0, "currentStep"].%X26 )
      Coil( "outputs".activeMask[26] )
   END_RUNG
   RUNG wire#powerrail
      Contact( "outputs".maskSequence[0, "currentStep"].%X27 )
      Coil( "outputs".activeMask[27] )
   END_RUNG
   RUNG wire#powerrail
      Contact( "outputs".maskSequence[0, "currentStep"].%X28 )
      Coil( "outputs".activeMask[28] )
   END_RUNG
   RUNG wire#powerrail
      Contact( "outputs".maskSequence[0, "currentStep"].%X29 )
      Coil( "outputs".activeMask[29] )
   END_RUNG
   RUNG wire#powerrail
      Contact( "outputs".maskSequence[0, "currentStep"].%X30 )
      Coil( "outputs".activeMask[30] )
   END_RUNG
   RUNG wire#powerrail
      Contact( "outputs".maskSequence[0, "currentStep"].%X31 )
      Coil( "outputs".activeMask[31] )
   END_RUNG
   // the same network as SCL:
   "outputs".activeMask[0] := "outputs".maskSequence[0, "currentStep"].%X0;
   "outputs".activeMask[1] := "outputs".maskSequence[0, "currentStep"].%X1;
   "outputs".activeMask[2] := "outputs".maskSequence[0, "currentStep"].%X2;
   "outputs".activeMask[3] := "outputs".maskSequence[0, "currentStep"].%X3;
   "outputs".activeMask[4] := "outputs".maskSequence[0, "currentStep"].%X4;
   "outputs".activeMask[5] := "outputs".maskSequence[0, "currentStep"].%X5;
   "outputs".activeMask[6] := "outputs".maskSequence[0, "currentStep"].%X6;
   "outputs".activeMask[7] := "outputs".maskSequence[0, "currentStep"].%X7;
   "outputs".activeMask[8] := "outputs".maskSequence[0, "currentStep"].%X8;
   "outputs".activeMask[9] := "outputs".maskSequence[0, "currentStep"].%X9;
   "outputs".activeMask[10] := "outputs".maskSequence[0, "currentStep"].%X10;
   "outputs".activeMask[11] := "outputs".maskSequence[0, "currentStep"].%X11;
   "outputs".activeMask[12] := "outputs".maskSequence[0, "currentStep"].%X12;
   "outputs".activeMask[13] := "outputs".maskSequence[0, "currentStep"].%X13;
   "outputs".activeMask[14] := "outputs".maskSequence[0, "currentStep"].%X14;
   "outputs".activeMask[15] := "outputs".maskSequence[0, "currentStep"].%X15;
   "outputs".activeMask[16] := "outputs".maskSequence[0, "currentStep"].%X16;
   "outputs".activeMask[17] := "outputs".maskSequence[0, "currentStep"].%X17;
   "outputs".activeMask[18] := "outputs".maskSequence[0, "currentStep"].%X18;
   "outputs".activeMask[19] := "outputs".maskSequence[0, "currentStep"].%X19;
   "outputs".activeMask[20] := "outputs".maskSequence[0, "currentStep"].%X20;
   "outputs".activeMask[21] := "outputs".maskSequence[0, "currentStep"].%X21;
   "outputs".activeMask[22] := "outputs".maskSequence[0, "currentStep"].%X22;
   "outputs".activeMask[23] := "outputs".maskSequence[0, "currentStep"].%X23;
   "outputs".activeMask[24] := "outputs".maskSequence[0, "currentStep"].%X24;
   "outputs".activeMask[25] := "outputs".maskSequence[0, "currentStep"].%X25;
   "outputs".activeMask[26] := "outputs".maskSequence[0, "currentStep"].%X26;
   "outputs".activeMask[27] := "outputs".maskSequence[0, "currentStep"].%X27;
   "outputs".activeMask[28] := "outputs".maskSequence[0, "currentStep"].%X28;
   "outputs".activeMask[29] := "outputs".maskSequence[0, "currentStep"].%X29;
   "outputs".activeMask[30] := "outputs".maskSequence[0, "currentStep"].%X30;
   "outputs".activeMask[31] := "outputs".maskSequence[0, "currentStep"].%X31;
END_REGION
END_FUNCTION
